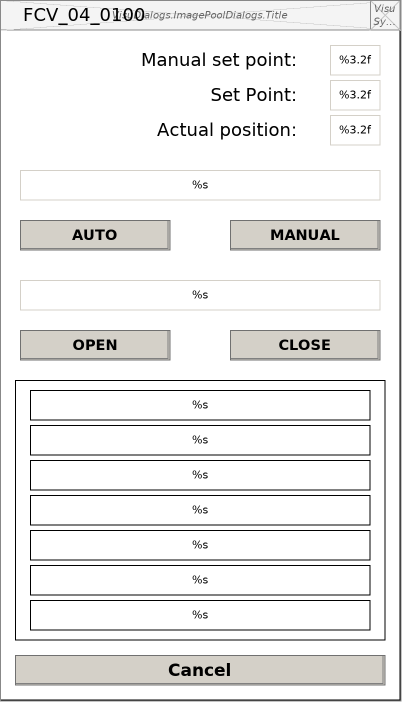
VISUALIZATION visuFCVDiag  // 402x702
    Rectangle (0,0 400x700)
    Button (20,220 150x30), "AUTO"
        tap progFCVCntrl.FCV_04_0100.AutoReq
    Button (230,220 150x30), "MANUAL"
        tap progFCVCntrl.FCV_04_0100.ManReq
    Button (20,330 150x30), "OPEN"
        tap progFCVCntrl.FCV_04_0100.ManOpenReq
    Button (230,330 150x30), "CLOSE"
        tap progFCVCntrl.FCV_04_0100.ManCloseReq
    Textfield (20,170 360x30), "%s", text variable: progFCVCntrl.FCV_04_0100.strAutoMan
    Textfield (20,280 360x30), "%s", text variable: progFCVCntrl.FCV_04_0100.strOpenTravClose
    Image (0,0 400x30), image: VisuDialogs.ImagePoolDialogs.Title
    Group (370,0 30x30)
        RoundedRectangle (0,0 30x30)
        Image (0,0 30x30), image: VisuSymbols.Symbols.Wrong
    Rectangle (15,380 370x260)
    RoundedRectangle (30,390 340x30), "%s", text variable: progFCVCntrl.FCV_04_0100.strInterlock_1
    RoundedRectangle (30,425 340x30), "%s", text variable: progFCVCntrl.FCV_04_0100.strInterlock_2
    RoundedRectangle (30,460 340x30), "%s", text variable: progFCVCntrl.FCV_04_0100.strInterlock_3
    RoundedRectangle (30,495 340x30), "%s", text variable: progFCVCntrl.FCV_04_0100.strInterlock_4
    RoundedRectangle (30,530 340x30), "%s", text variable: progFCVCntrl.FCV_04_0100.strInterlock_5
    RoundedRectangle (30,565 340x30), "%s", text variable: progFCVCntrl.FCV_04_0100.strInterlock_6
    RoundedRectangle (30,600 340x30), "%s", text variable: progFCVCntrl.FCV_04_0100.strInterlock_7
    Button (15,655 370x30), "Cancel"
    Label (0,80 300x30), "Set Point:"
    Textfield (330,80 50x30), "%3.2f", text variable: progFCVCntrl.FCV_04_0100.CmdSpOut
    Label (0,45 300x30), "Manual set point:"
    Textfield (330,45 50x30), "%3.2f", text variable: progFCVCntrl.FCV_04_0100.ManSP
        OnMouseClick: write progFCVCntrl.FCV_04_0100.ManSP via VisuDialogs.NumpadExtended
    Label (0,115 300x30), "Actual position:"
    Textfield (330,115 50x30), "%3.2f", text variable: progFCVCntrl.FCV_04_0100.ActPos
    Label (20,0 210x30), "FCV_04_0100"
END_VISUALIZATION

(* stored: Version 1.1.0.1, ProductVersion 3.1.4022.17
   Visu visuFCVDiag: Id {470414b8-0e39-45ee-8187-ffb075db576a} *)
